//{attribute 'qualified_only'}
VAR_GLOBAL
	TxBufferTB : ComBuffer; (* Receive data buffer; used with all receive function blocks *)
	RxBufferTB : ComBuffer; (* Transmit data buffer; used with all receive function blocks *)
	
	TxBufferLH : ComBuffer; //잘동작되면 TB도 지역변수로 변경
	RxBufferLH : ComBuffer;	
END_VAR

(* stored: Version 1.1.0.1, ProductVersion 3.1.4024.12
   GVL GVL_Serial: Id {2f04b256-d3e9-429e-bb30-15aa5e82ca02} *)
